FUNCTION_BLOCK FINAL Signal IMPLEMENTS I_SignalNode, I_Signal
VAR
	_fbTag			: Tags.Tag;
	_nCount			: UDINT;
	_nSize			: UDINT;
	_nId			: UDINT;
END_VAR

PROPERTY INTERNAL count : UDINT
GET
count := _nCount;
END_GET
SET
_nCount := count;
END_SET
END_PROPERTY

METHOD Emit
VAR_INPUT
	iTag			: Tags.I_Tag := 0;
END_VAR
IF iTag = 0 THEN
	iTag := _fbTag;
END_IF

_EmitSignal(THIS^, iTag);
END_METHOD

PROPERTY INTERNAL id : UDINT
GET
id := _nId;
END_GET
SET
_nId := id;
END_SET
END_PROPERTY

METHOD Option : REFERENCE TO Signal
VAR_INPUT
	sOption		: Strings.Str;
END_VAR
Option REF= THIS^;
_fbTag.Option := sOption;
END_METHOD

METHOD Pair : Results.Result
VAR_INPUT
	iReceiver		: I_Receiver;
END_VAR
IF iReceiver = 0 THEN
	Pair := Results.Err.Itf0;
ELSIF iReceiver.IsOk THEN
	Pair := _NewPair(THIS^, iReceiver);
ELSE
	Pair := Results.Error;
END_IF
END_METHOD

PROPERTY INTERNAL size : UDINT
GET
size := _nSize;
END_GET
SET
_nSize := size;
END_SET
END_PROPERTY

PROPERTY Tag : Tags.I_Tag
GET
Tag := _fbTag;
END_GET
END_PROPERTY

METHOD ToDebug : Debug.I_Debug
ToDebug := THIS^;
END_METHOD

METHOD Unpair : Results.Result
VAR_INPUT
	iReceiver		: I_Receiver;
END_VAR
IF iReceiver = 0 THEN
	Unpair := Results.Err.Itf0;
ELSIF iReceiver.IsOk THEN
	Unpair := _Unpair(THIS^, iReceiver);
ELSE
	Unpair := Results.Error;
END_IF
END_METHOD

END_FUNCTION_BLOCK

(* stored: Version 1.1.0.1
   POU Signal: Id {7c9b617f-f7bd-442d-b8c9-34e8d7bdc353}, SpecialFunc None
   Folder Node: Id {1c06cc1f-8118-48fe-8ba5-55eb66c8e846}
   Property count: Id {f0af54fa-0857-4928-a20f-0a9e19647f93}
   Get Get: Id {b3963a5f-a76a-43cc-96e4-af6f9e4e44c2}
   Set Set: Id {c04c49b1-c4c3-4704-bb39-a536cd6f73f3}
   Method Emit: Id {d0827b51-da6b-4d29-b0a4-e9daca3aa340}
   Property id: Id {819ef4a3-3ea7-4562-a22a-db3e51f6c5da}
   Get Get: Id {f016ae8a-7c20-4ce4-9027-82c29b8cabd2}
   Set Set: Id {95c075e4-42b4-442d-82bf-ffe4e4510c79}
   Method Option: Id {0ff0a38b-8cae-4a43-a082-d0a5b09641ff}
   Method Pair: Id {d45162d9-176c-4304-b03f-8a4e26d88ae6}
   Property size: Id {99f5d688-c7d1-4660-8e05-53b7b2f0a0b8}
   Get Get: Id {480c9fec-29fc-4477-9608-0888d461f887}
   Set Set: Id {68795c0e-0755-495b-8c14-44aca974c6e1}
   Property Tag: Id {ae8fb298-bf52-4d66-bee9-240c71f53a49}
   Get Get: Id {7858a5b1-6904-4110-a1d7-ec2262f1063e}
   Method ToDebug: Id {2366606e-7015-468b-a9e3-80d32e0b5814}
   Method Unpair: Id {ae27d934-17a9-4eae-a002-1ba80dc83d65} *)
